// TIA Portal project "0000" (V15.1)

(* hardware
DEVICE "S7-1200-Station_1"  S7-1200 Station
   slot 0: "Baugruppenträger_0"  S7-1200 Rack  Rack  V1.0
   slot 1: "0000"  CPU 1214C DC/DC/DC  6ES7 214-1AG40-0XB0  V4.3
DEVICE "S7300/ET200M-Station_1"  S7-300 station
   slot 0: "Profilschiene_0"  Rail  6ES7 390-1***0-0AA0
   slot 2: "0001"  CPU 317-2 PN/DP  6ES7 317-2EK13-0AB0  V2.6
      slot 1: "MPI/DP-Schnittstelle_1"  X1
      slot 2: "PROFINET-Schnittstelle_1"  PN-IO
         slot 1: "Port_1"  Port
DEVICE "S71500/ET200MP-Station_1"  S7-1500 station
   slot 0: "Profilschiene_0"  Rack  6ES7 590-1***0-0AA0
   slot 1: "PLC_1"  CPU 1515-2 PN  6ES7 515-2AM01-0AB0  V2.6
      slot 3: "CPU-Display_1"  6ES7591-1BA00-0AA0
*)

// ===== PLC "0000"  CPU 1214C DC/DC/DC =====

VAR_GLOBAL   // PLC tag table "Standard-Variablentabelle"
   "Clock_Byte" AT %MB1 : Byte;
   "Clock_10Hz" AT %M1.0 : Bool;
   "Clock_5Hz" AT %M1.1 : Bool;
   "Clock_2.5Hz" AT %M1.2 : Bool;
   "Clock_2Hz" AT %M1.3 : Bool;
   "Clock_1.25Hz" AT %M1.4 : Bool;
   "Clock_1Hz" AT %M1.5 : Bool;
   "Clock_0.625Hz" AT %M1.6 : Bool;
   "Clock_0.5Hz" AT %M1.7 : Bool;
   "System_Byte" AT %MB0 : Byte;
   "FirstScan" AT %M0.0 : Bool;
   "DiagStatusUpdate" AT %M0.1 : Bool;
   "AlwaysTRUE" AT %M0.2 : Bool;
   "AlwaysFALSE" AT %M0.3 : Bool;
   "Test" AT %M10.0 : Bool;
   "Tag_1" AT %M100.0 : Bool;
   "Tag_2" AT %M100.2 : Bool;
   "Tag_3" AT %M200.0 : Bool;
   "%M200.1" AT %M200.1 : Bool;
END_VAR

TYPE "Daten"
TITLE = has no title
// some comment
   STRUCT
      Aktiv : Bool := True;   // Anlage an oder aus
      Codierung : Byte := 16#2;   // Codierung
      Status : Word := 16#FF;   // Status
      Status_erweitert : DWord := 16#FFFF;   // Erweiterter Status
      Programmnummer : Int := 3;   // Aktuelle Programmnummer
      Zaehler : DInt := 5;   // Zählerstand
      Stationsname : String := 'Anlage001';   // Name der Station
      Zeitstempel : DTL;   // Aktueller Zeitstempel
   END_STRUCT;
END_TYPE

DATA_BLOCK "ConPlc_DB"   // DB1
{ S7_Optimized_Access := 'TRUE' }
VERSION : 0.1
// stored: InstanceOfName ConPlc
"ConPlc"
BEGIN
END_DATA_BLOCK

// folder: Testdata

DATA_BLOCK "Testdata"   // DB3
{ S7_Optimized_Access := 'FALSE' }
VERSION : 0.1
   VAR
      Daten : "Daten";
   END_VAR
BEGIN
END_DATA_BLOCK

// folder: (top level)

FUNCTION_BLOCK "ConPlc"   // FB1000, SCL
{ S7_Optimized_Access := 'TRUE' }
VERSION : 0.1
   VAR_INPUT
      ACTIVATE : Bool := False;   // activate connection
      TACT : Bool := False;   // tact
      CONN_ID : Conn_Ouc := 16#1;   // connection reference / identifier
      HW_ID : Hw_Any := 64;   // HW-identifier of IE-interface submodule
      CONN_Type : Byte := 16#0B;   // type of connection: 11=TCP/IP, 19=UDP (17=TCP/IP)
      IP_ADDR_1 : Byte := 16#C0;   // IPv4 address
      IP_ADDR_2 : Byte := 16#A8;   // IPv4 address
      IP_ADDR_3 : Byte := 16#00;   // IPv4 address
      IP_ADDR_4 : Byte := 16#1E;   // IPv4 address
      PORT_Remote : UInt := 2000;   // remote UDP/TCP port number
      PORT_Local : UInt := 2000;   // local UDP/TCP port number
   END_VAR
   VAR_IN_OUT
      DATA : Variant;
   END_VAR
   VAR
      ACT_CONN : Bool;
      CONN_ESTABLISHED : Bool;
      DONE_CONN : Bool;
      BUSY_CONN : Bool;
      ERROR_CONN : Bool;
      STATUS_CONN : Word;
      DONE_SEND : Bool;
      BUSY_SEND : Bool;
      ERROR_SEND : Bool;
      STATUS_SEND : Word;
      ACT_SEND : Bool;
      NDR_RECV : Bool;
      BUSY_RECV : Bool;
      ERROR_RECV : Bool;
      STATUS_RECV : Word;
      RCVD_LEN : UDInt;
      ACT_RECV : Bool;
      DONE_DISCON : Bool;
      BUSY_DISCON : Bool;
      ERROR_DISCON : Bool;
      STATUS_DISCON : Word;
      ACT_DISCON : Bool;
      TRIGGER : Bool;
      TRIGGER_MEM : Bool;
      TCON_IDB : TCON;
      TSEND_IDB : TSEND;
      TRCV_IDB : TRCV;
      TDISCON_IDB : TDISCON;
      CONN_PARAMETER : TCON_IP_v4;
      TON_RESET : TON_TIME;
   END_VAR
   // CONN_PARAMETER.InterfaceId := 64;
   // CONN_PARAMETER.ID := 16#1;
   // CONN_PARAMETER.ConnectionType := 16#0B;
   // CONN_PARAMETER.ActiveEstablished := False;
   // CONN_PARAMETER.RemoteAddress.ADDR[1] := 16#C0;
   // CONN_PARAMETER.RemoteAddress.ADDR[2] := 16#A8;
   // CONN_PARAMETER.RemoteAddress.ADDR[3] := 16#00;
   // CONN_PARAMETER.RemoteAddress.ADDR[4] := 16#1E;
   // CONN_PARAMETER.RemotePort := 2000;
   // CONN_PARAMETER.LocalPort := 2000;
BEGIN
   REGION set connection data
       #CONN_PARAMETER.ID := #CONN_ID;
       #CONN_PARAMETER.InterfaceId := #HW_ID;
       #CONN_PARAMETER.ActiveEstablished := TRUE;
       #CONN_PARAMETER.ConnectionType := #CONN_Type;
       #CONN_PARAMETER.RemoteAddress.ADDR[1] := #IP_ADDR_1;
       #CONN_PARAMETER.RemoteAddress.ADDR[2] := #IP_ADDR_2;
       #CONN_PARAMETER.RemoteAddress.ADDR[3] := #IP_ADDR_3;
       #CONN_PARAMETER.RemoteAddress.ADDR[4] := #IP_ADDR_4;
       #CONN_PARAMETER.RemotePort := #PORT_Remote;
       #CONN_PARAMETER.LocalPort := #PORT_Local;
   END_REGION

   REGION create trigger
       #TRIGGER := #TACT AND NOT #TRIGGER_MEM;
       #TRIGGER_MEM := #TACT;
   END_REGION

   REGION connect
       //connect enable
       IF #ACTIVATE AND NOT #CONN_ESTABLISHED THEN
           #ACT_CONN := True;
       END_IF;
       //connect
       #TCON_IDB(REQ       := #ACT_CONN AND #TRIGGER,
                 ID        := #CONN_ID,
                 DONE      => #DONE_CONN,
                 BUSY      => #BUSY_CONN,
                 ERROR     => #ERROR_CONN,
                 STATUS    => #STATUS_CONN,
                 CONNECT   := #CONN_PARAMETER);
       //connect done
       IF #DONE_CONN THEN
           #CONN_ESTABLISHED := True;
           #ACT_CONN := False;
       END_IF;
   END_REGION

   REGION send
       //send enable
       #ACT_SEND := #CONN_ESTABLISHED AND #TRIGGER AND NOT #BUSY_SEND;
       //send
       #TSEND_IDB(REQ      := #ACT_SEND,
                  ID       := #CONN_ID,
                  LEN      := 0,
                  DONE     => #DONE_SEND,
                  BUSY     => #BUSY_SEND,
                  ERROR    => #ERROR_SEND,
                  STATUS   => #STATUS_SEND,
                  DATA     := #DATA);
   END_REGION

   // REGION recieve
   //     //revieve enable
   //     #ACT_RECV := #CONN_ESTABLISHED;
   //     //recieve
   //     #TRCV_IDB(EN_R      := #ACT_RECV,
   //               ID        := #CONN_ID,
   //               LEN       := 0,
   //               ADHOC     := FALSE,
   //               NDR       => #NDR_RECV,
   //               BUSY      => #BUSY_RECV,
   //               ERROR     => #ERROR_RECV,
   //               STATUS    => #STATUS_RECV,
   //               RCVD_LEN  => #RCVD_LEN,
   //               DATA      := #DATA);
   // END_REGION

   REGION disconnect
       //disconnect enable
       #TON_RESET(IN := #ACTIVATE AND NOT #CONN_ESTABLISHED,
                  PT := T#5s);
       #ACT_DISCON := (#TON_RESET.Q) OR (NOT #ACTIVATE);
       //disconnect
       #TDISCON_IDB(REQ    := #ACT_DISCON,
                    ID     := #CONN_ID,
                    DONE   => #DONE_DISCON,
                    BUSY   => #BUSY_DISCON,
                    ERROR  => #ERROR_DISCON,
                    STATUS => #STATUS_DISCON);

       //disconnect done
       IF NOT #ACTIVATE THEN
           #CONN_ESTABLISHED := False;
           #ACT_CONN := False;
       END_IF;
   END_REGION
END_FUNCTION_BLOCK

ORGANIZATION_BLOCK "Main"   // OB1, FBD, ProgramCycle
TITLE = "Main Program Sweep (Cycle)"
{ S7_Optimized_Access := 'TRUE' }
VERSION : 0.1
   VAR_INPUT
      Initial_Call : Bool;   // Initial call of this OB
      Remanence : Bool;   // =True, if remanent data are available
   END_VAR
   VAR_TEMP
      retval : Int;
   END_VAR
BEGIN

REGION Network 1
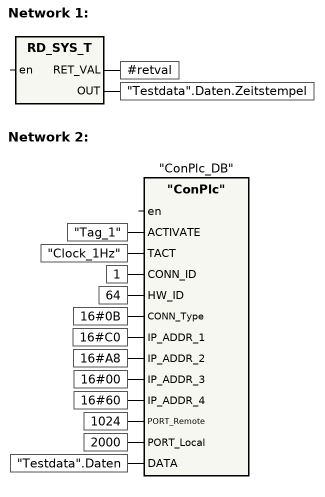
   #retval := RD_SYS_T(OUT => "Testdata".Daten.Zeitstempel);
END_REGION

REGION Network 2
   "ConPlc_DB"(ACTIVATE := "Tag_1",   // "ConPlc"
               TACT := "Clock_1Hz",
               CONN_ID := 1,
               HW_ID := 64,
               CONN_Type := 16#0B,
               IP_ADDR_1 := 16#C0,
               IP_ADDR_2 := 16#A8,
               IP_ADDR_3 := 16#00,
               IP_ADDR_4 := 16#60,
               PORT_Remote := 1024,
               PORT_Local := 2000,
               DATA := "Testdata".Daten);
END_REGION
END_ORGANIZATION_BLOCK

// ===== PLC "0001"  CPU 317-2 PN/DP =====

VAR_GLOBAL   // PLC tag table "Standard-Variablentabelle"
   "Test" AT %M10.0 : Bool;
   "Clock_Byte" AT %MB0 : Byte;
   "Clock_10Hz" AT %M0.0 : Bool;
   "Clock_5Hz" AT %M0.1 : Bool;
   "Clock_2.5Hz" AT %M0.2 : Bool;
   "Clock_2Hz" AT %M0.3 : Bool;
   "Clock_1.25Hz" AT %M0.4 : Bool;
   "Clock_1Hz" AT %M0.5 : Bool;
   "Clock_0.625Hz" AT %M0.6 : Bool;
   "Clock_0.5Hz" AT %M0.7 : Bool;
END_VAR

ORGANIZATION_BLOCK "Main"   // OB1, SCL
TITLE = "Main Program Sweep (Cycle)"
{ S7_Optimized_Access := 'FALSE' }
VERSION : 0.1
   VAR_TEMP
      OB1_EV_CLASS : Byte;   // Bits 0-3 = 1 (Coming event), Bits 4-7 = 1 (Event class 1)
      OB1_SCAN_1 : Byte;   // 1 (Cold restart scan 1 of OB 1), 3 (Scan 2-n of OB 1)
      OB1_PRIORITY : Byte;   // Priority of OB Execution
      OB1_OB_NUMBR : Byte;   // 1 (Organization block 1, OB1)
      OB1_RESERVED_1 : Byte;   // Reserved for system
      OB1_RESERVED_2 : Byte;   // Reserved for system
      OB1_PREV_CYCLE : Int;   // Cycle time of previous OB1 scan (milliseconds)
      OB1_MIN_CYCLE : Int;   // Minimum cycle time of OB1 (milliseconds)
      OB1_MAX_CYCLE : Int;   // Maximum cycle time of OB1 (milliseconds)
      OB1_DATE_TIME : Date_And_Time;   // Date and time OB1 started
   END_VAR
BEGIN
   REGION Test
       "Test" := "Clock_0.5Hz";
   END_REGION
END_ORGANIZATION_BLOCK

// ===== PLC "PLC_1"  CPU 1515-2 PN =====

FUNCTION_BLOCK "S7-1500_CPU_Comm_TCP_master"   // FB250, STL
TITLE = FB to master connection to partner CPU
{ S7_Optimized_Access := 'FALSE' }
VERSION : 0.1
   VAR_INPUT
      CONN_stop : Bool := False;   // stop connection
      Takt : Bool := False;
      CONN_ID : Conn_Ouc := 16#1;   // connection reference / identifier
      HW_ID : Hw_Any := 64;   // HW-identifier of IE-interface submodule
      CONN_Type : Byte := 16#0B;   // type of connection: 11=TCP/IP, 19=UDP (17=TCP/IP)
      IP_ADDR_1 : Byte := 16#C0;   // IPv4 address
      IP_ADDR_2 : Byte := 16#A8;   // IPv4 address
      IP_ADDR_3 : Byte := 16#00;   // IPv4 address
      IP_ADDR_4 : Byte := 16#1E;   // IPv4 address
      remote_port : UInt := 2000;   // remote UDP/TCP port number
      local_port : UInt := 2000;   // local UDP/TCP port number
   END_VAR
   VAR
      START_CONN : Bool;
      CONN_established : Bool;
      DONE_CONN : Bool;
      BUSY_CONN : Bool;
      ERROR_CONN : Bool;
      STATUS_CONN : Word;
      DONE_SEND : Bool;
      BUSY_SEND : Bool;
      ERROR_SEND : Bool;
      STATUS_SEND : Word;
      ACT_SEND : Bool;
      NDR_RECV : Bool;
      BUSY_RECV : Bool;
      ERROR_RECV : Bool;
      STATUS_RECV : Word;
      RCVD_LEN : UDInt;
      DONE_DISCON : Bool;
      BUSY_DISCON : Bool;
      ERROR_DISCON : Bool;
      STATUS_DISCON : Word;
      TCON_IDB : TCON;
      TSEND_IDB : TSEND;
      TRCV_IDB : TRCV;
      TDISCON_IDB : TDISCON;
      CONN_parameter : TCON_IP_v4;
      SEND_DATA : Struct
         Lebensbit : Bool;
         Störung_Vakuum : Bool;
         Reserve_bit_2 : Bool;
         Reserve_bit_3 : Bool;
         Reserve_bit_4 : Bool;
         Reserve_bit_5 : Bool;
         Reserve_bit_6 : Bool;
         Reserve_bit_7 : Bool;
         Temperatur : Int := 20;   // Umgebungstemperatur in °C
         Absolutdruck : Int := 1000;   // Absolutdruck in mbar
      END_STRUCT;
      RECV_DATA : Struct
         Lebensbit : Bool;
         Reserve_bit_1 : Bool;
         Reserve_bit_2 : Bool;
         Reserve_bit_3 : Bool;
         Reserve_bit_4 : Bool;
         Reserve_bit_5 : Bool;
         Reserve_bit_6 : Bool;
         Reserve_bit_7 : Bool;
      END_STRUCT;
   END_VAR
   VAR_TEMP
      conn_trigger : Bool;
   END_VAR
   // CONN_parameter.InterfaceId := 64;
   // CONN_parameter.ID := 16#1;
   // CONN_parameter.ConnectionType := 16#0B;
   // CONN_parameter.ActiveEstablished := False;
   // CONN_parameter.RemotePort := 2000;
   // CONN_parameter.LocalPort := 2000;
   // CONN_parameter.RemoteAddress.ADDR[1] := 16#C0;
   // CONN_parameter.RemoteAddress.ADDR[2] := 16#A8;
   // CONN_parameter.RemoteAddress.ADDR[3] := 16#00;
   // CONN_parameter.RemoteAddress.ADDR[4] := 16#1E;
BEGIN

REGION Network 1: set connection data
   //---------------------------------
         L     #CONN_ID;
         T     #CONN_parameter.ID;
   //---------------------------------
         L     #HW_ID;
         T     #CONN_parameter.InterfaceId;
   //---------------------------------
         SET;  //Master wartet das sich der slave meldet
         R     #CONN_parameter.ActiveEstablished;
   //---------------------------------
         L     #CONN_Type;
         T     #CONN_parameter.ConnectionType;
   //---------------------------------
         L     #IP_ADDR_1;
         T     #CONN_parameter.RemoteAddress.ADDR[1];
         L     #IP_ADDR_2;
         T     #CONN_parameter.RemoteAddress.ADDR[2];
         L     #IP_ADDR_3;
         T     #CONN_parameter.RemoteAddress.ADDR[3];
         L     #IP_ADDR_4;
         T     #CONN_parameter.RemoteAddress.ADDR[4];
   //---------------------------------
         L     #remote_port;
         T     #CONN_parameter.RemotePort;
   //---------------------------------
         L     #local_port;
         T     #CONN_parameter.LocalPort;
   //---------------------------------
END_REGION

REGION Network 2: start connect
         A(;
         AN    #CONN_established;
         AN    #CONN_stop;
         );
         S     #START_CONN;
END_REGION

REGION Network 3: connect
         A     #START_CONN;
         =     #conn_trigger;

         CALL  #TCON_IDB
         ( REQ     := #conn_trigger,
           ID      := #CONN_ID,
           DONE    := #DONE_CONN,
           BUSY    := #BUSY_CONN,
           ERROR   := #ERROR_CONN,
           STATUS  := #STATUS_CONN,
           CONNECT := #CONN_parameter
         );
END_REGION

REGION Network 4: done connect
         A     #DONE_CONN;
         S     #CONN_established;
         R     #START_CONN;
END_REGION

REGION Network 5: automaticly trigger send data if sending is not active anymore
         AN    #BUSY_SEND;
         A     #Takt;
         =     #ACT_SEND;
END_REGION

REGION Network 6: send
         CALL  #TSEND_IDB
         ( REQ    := #ACT_SEND,
           ID     := #CONN_ID,
           LEN    := 0,
           DONE   := #DONE_SEND,
           BUSY   := #BUSY_SEND,
           ERROR  := #ERROR_SEND,
           STATUS := #STATUS_SEND,
           DATA   := #SEND_DATA
         );
END_REGION

REGION Network 7: recieve
         CALL  #TRCV_IDB
         ( EN_R     := #CONN_established,
           ID       := #CONN_ID,
           LEN      := 0,
           ADHOC    := FALSE,
           NDR      := #NDR_RECV,
           BUSY     := #BUSY_RECV,
           ERROR    := #ERROR_RECV,
           STATUS   := #STATUS_RECV,
           RCVD_LEN := #RCVD_LEN,
           DATA     := #RECV_DATA
         );
END_REGION

REGION Network 8: disconnect
         A     #CONN_stop;
         R     #CONN_established;
         R     #START_CONN;

         CALL  #TDISCON_IDB
         ( REQ    := #CONN_stop,
           ID     := #CONN_ID,
           DONE   := #DONE_DISCON,
           BUSY   := #BUSY_DISCON,
           ERROR  := #ERROR_DISCON,
           STATUS := #STATUS_DISCON
         );
END_REGION
END_FUNCTION_BLOCK

FUNCTION_BLOCK "S7-1500_CPU_Comm_TCP_slave"   // FB251, STL
TITLE = FB to slave connection to partner CPU
{ S7_Optimized_Access := 'FALSE' }
VERSION : 0.1
   VAR_INPUT
      CONN_stop : Bool := False;   // stop connection
      Takt : Bool := False;
      CONN_ID : Conn_Ouc := 16#1;   // connection reference / identifier
      HW_ID : Hw_Any := 64;   // HW-identifier of IE-interface submodule
      CONN_Type : Byte := 16#0B;   // type of connection: 11=TCP/IP, 19=UDP (17=TCP/IP)
      IP_ADDR_1 : Byte := 16#C0;   // IPv4 address
      IP_ADDR_2 : Byte := 16#A8;   // IPv4 address
      IP_ADDR_3 : Byte := 16#00;   // IPv4 address
      IP_ADDR_4 : Byte := 16#1E;   // IPv4 address
      remote_port : UInt := 2000;   // remote UDP/TCP port number
      local_port : UInt := 2000;   // local UDP/TCP port number
   END_VAR
   VAR
      START_CONN : Bool;
      CONN_established : Bool;
      DONE_CONN : Bool;
      BUSY_CONN : Bool;
      ERROR_CONN : Bool;
      STATUS_CONN : Word;
      DONE_SEND : Bool;
      BUSY_SEND : Bool;
      ERROR_SEND : Bool;
      STATUS_SEND : Word;
      ACT_SEND : Bool;
      NDR_RECV : Bool;
      BUSY_RECV : Bool;
      ERROR_RECV : Bool;
      STATUS_RECV : Word;
      RCVD_LEN : UDInt;
      DONE_DISCON : Bool;
      BUSY_DISCON : Bool;
      ERROR_DISCON : Bool;
      STATUS_DISCON : Word;
      TCON_IDB : TCON;
      TSEND_IDB : TSEND;
      TRCV_IDB : TRCV;
      TDISCON_IDB : TDISCON;
      CONN_parameter : TCON_IP_v4;
      SEND_DATA : Struct
         Lebensbit : Bool;
         Reserve_bit_1 : Bool;
         Reserve_bit_2 : Bool;
         Reserve_bit_3 : Bool;
         Reserve_bit_4 : Bool;
         Reserve_bit_5 : Bool;
         Reserve_bit_6 : Bool;
         Reserve_bit_7 : Bool;
      END_STRUCT;
      RECV_DATA : Struct
         Lebensbit : Bool;
         Störung_Vakuum : Bool;
         Reserve_bit_2 : Bool;
         Reserve_bit_3 : Bool;
         Reserve_bit_4 : Bool;
         Reserve_bit_5 : Bool;
         Reserve_bit_6 : Bool;
         Reserve_bit_7 : Bool;
         Temperatur : Int := 20;   // Umgebungstemperatur in °C
         Absolutdruck : Int := 1000;   // Absolutdruck in mbar
      END_STRUCT;
   END_VAR
   VAR_TEMP
      conn_trigger : Bool;
   END_VAR
   // CONN_parameter.InterfaceId := 64;
   // CONN_parameter.ID := 16#1;
   // CONN_parameter.ConnectionType := 16#0B;
   // CONN_parameter.ActiveEstablished := False;
   // CONN_parameter.RemotePort := 2000;
   // CONN_parameter.LocalPort := 2000;
   // CONN_parameter.RemoteAddress.ADDR[1] := 16#C0;
   // CONN_parameter.RemoteAddress.ADDR[2] := 16#A8;
   // CONN_parameter.RemoteAddress.ADDR[3] := 16#00;
   // CONN_parameter.RemoteAddress.ADDR[4] := 16#1E;
BEGIN

REGION Network 1: xxxset connection data
   //---------------------------------
         L     #CONN_ID;
         T     #CONN_parameter.ID;
   //---------------------------------
         L     #HW_ID;
         T     #CONN_parameter.InterfaceId;
   //---------------------------------
         SET;  //Slave versucht aktiv die verbindung aufzubauen
         S     #CONN_parameter.ActiveEstablished;
   //---------------------------------
         L     #CONN_Type;
         T     #CONN_parameter.ConnectionType;
   //---------------------------------
         L     #IP_ADDR_1;
         T     #CONN_parameter.RemoteAddress.ADDR[1];
         L     #IP_ADDR_2;
         T     #CONN_parameter.RemoteAddress.ADDR[2];
         L     #IP_ADDR_3;
         T     #CONN_parameter.RemoteAddress.ADDR[3];
         L     #IP_ADDR_4;
         T     #CONN_parameter.RemoteAddress.ADDR[4];
   //---------------------------------
         L     #remote_port;
         T     #CONN_parameter.RemotePort;
   //---------------------------------
         L     #local_port;
         T     #CONN_parameter.LocalPort;
   //---------------------------------
END_REGION

REGION Network 2: xxxstart connect
         A(;
         AN    #CONN_established;
         AN    #CONN_stop;
         );
         S     #START_CONN;
END_REGION

REGION Network 3: xxxconnect
         A     #START_CONN;
         A     #Takt;
         =     #conn_trigger;

         CALL  #TCON_IDB
         ( REQ     := #conn_trigger,
           ID      := #CONN_ID,
           DONE    := #DONE_CONN,
           BUSY    := #BUSY_CONN,
           ERROR   := #ERROR_CONN,
           STATUS  := #STATUS_CONN,
           CONNECT := #CONN_parameter
         );
END_REGION

REGION Network 4: xxxdone connect
         A     #DONE_CONN;
         S     #CONN_established;
         R     #START_CONN;
END_REGION

REGION Network 5: automaticly trigger send data if new data recieved
         A     #NDR_RECV;
         =     #ACT_SEND;
END_REGION

REGION Network 6: send
         CALL  #TSEND_IDB
         ( REQ    := #ACT_SEND,
           ID     := #CONN_ID,
           LEN    := 0,
           DONE   := #DONE_SEND,
           BUSY   := #BUSY_SEND,
           ERROR  := #ERROR_SEND,
           STATUS := #STATUS_SEND,
           DATA   := #SEND_DATA
         );
END_REGION

REGION Network 7: recieve
         CALL  #TRCV_IDB
         ( EN_R     := #CONN_established,
           ID       := #CONN_ID,
           LEN      := 0,
           ADHOC    := FALSE,
           NDR      := #NDR_RECV,
           BUSY     := #BUSY_RECV,
           ERROR    := #ERROR_RECV,
           STATUS   := #STATUS_RECV,
           RCVD_LEN := #RCVD_LEN,
           DATA     := #RECV_DATA
         );
END_REGION

REGION Network 8: disconnect
         A     #CONN_stop;
         R     #CONN_established;
         R     #START_CONN;

         CALL  #TDISCON_IDB
         ( REQ    := #CONN_stop,
           ID     := #CONN_ID,
           DONE   := #DONE_DISCON,
           BUSY   := #BUSY_DISCON,
           ERROR  := #ERROR_DISCON,
           STATUS := #STATUS_DISCON
         );
END_REGION
END_FUNCTION_BLOCK

FUNCTION "SPS-Kommunikation" : Void   // FC250, STL
TITLE = Kommunikation mit anderer CPU aufbauen
{ S7_Optimized_Access := 'TRUE' }
VERSION : 0.1
   VAR_TEMP
      connection_stop : Bool;
   END_VAR
BEGIN

REGION Network 1: Daten rangieren
         L     "DB350_Umgebungseinflüsse".Temperatur;
         T     "S7-1500_CPU_Comm_TCP_master_DB".SEND_DATA.Temperatur;

         L     "DB350_Umgebungseinflüsse".Absolutdruck;
         T     "S7-1500_CPU_Comm_TCP_master_DB".SEND_DATA.Absolutdruck;

         A     "Störung_Vakuum";
         =     "S7-1500_CPU_Comm_TCP_master_DB".SEND_DATA.Störung_Vakuum;
END_REGION

REGION Network 2: Lebensbit mit Takt an Partner senden, Lebensbit von Partner überwachen
         A     "Clock_1Hz";
         =     "S7-1500_CPU_Comm_TCP_master_DB".SEND_DATA.Lebensbit;

         A     "ME_STSP_EIN";
         A     "S7-1500_CPU_Comm_TCP_master_DB".RECV_DATA.Lebensbit;
         L     s5t#10s;
         SD    "T-CPU-CPU_Comm_Error_01";

         A     "ME_STSP_EIN";
         AN    "S7-1500_CPU_Comm_TCP_master_DB".RECV_DATA.Lebensbit;
         L     s5t#10s;
         SD    "T-CPU-CPU_Comm_Error_02";
END_REGION

REGION Network 3: Kommunikationsaufruf
         A     "ME_STSP_EIN";
         L     s5t#3s;
         SE    "T-comm_restart";

         A     "T-comm_restart";
         =     #connection_stop;

   //CPU mit aktiven Verbindungsaufbau
         CALL  "S7-1500_CPU_Comm_TCP_master", "S7-1500_CPU_Comm_TCP_master_DB"
         ( CONN_stop   := #connection_stop,  //Stoppen der Verbindung
           Takt        := "Clock_0.5Hz",  //Taktsignal
           CONN_ID     := 5,
           HW_ID       := 64,  //HW-ID der Profinet Schnittstelle (in diesem Beispiel [X1])
           CONN_Type   := 16#0B,  //Steht für TCP verbindungsart
           IP_ADDR_1   := 16#C0,  //192 IP-Adresse der Partner CPU
           IP_ADDR_2   := 16#A8,  //168
           IP_ADDR_3   := 16#00,  //0
           IP_ADDR_4   := 16#04,  //4
           remote_port := 2000,  //partner Portnummer
           local_port  := 2000  //eigene Portnummer
         );
END_REGION
END_FUNCTION

FUNCTION "SPS-Kommunikation_1" : Void   // FC250, STL
TITLE = Kommunikation mit anderer CPU aufbauen
{ S7_Optimized_Access := 'TRUE' }
VERSION : 0.1
   VAR_TEMP
      connection_stop : Bool;
   END_VAR
BEGIN

REGION Network 1: Daten rangieren
         L     "S7-1500_CPU_Comm_TCP_slave_DB".RECV_DATA.Temperatur;
         T     "DB350_Umgebungseinflüsse".Temperatur;

         L     "S7-1500_CPU_Comm_TCP_slave_DB".RECV_DATA.Absolutdruck;
         T     "DB350_Umgebungseinflüsse".Absolutdruck;

         A     "S7-1500_CPU_Comm_TCP_slave_DB".RECV_DATA.Störung_Vakuum;
         =     "Störung_Vakuum";
END_REGION

REGION Network 2: Lebensbit mit Takt an Partner senden, Lebensbit von Partner überwachen
         A     "Clock_1Hz";
         =     "S7-1500_CPU_Comm_TCP_slave_DB".SEND_DATA.Lebensbit;

         A     "ME_STSP_EIN";
         A     "S7-1500_CPU_Comm_TCP_slave_DB".RECV_DATA.Lebensbit;
         L     s5t#10s;
         SD    "T-CPU-CPU_Comm_Error_01";

         A     "ME_STSP_EIN";
         AN    "S7-1500_CPU_Comm_TCP_slave_DB".RECV_DATA.Lebensbit;
         L     s5t#10s;
         SD    "T-CPU-CPU_Comm_Error_02";
END_REGION

REGION Network 3: Kommunikationsaufruf
         A     "ME_STSP_EIN";
         L     s5t#3s;
         SE    "T-comm_restart";

         A     "T-comm_restart";
         =     #connection_stop;

   //CPU mit Passivem Verbindungsaufbau
         CALL  "S7-1500_CPU_Comm_TCP_slave", "S7-1500_CPU_Comm_TCP_slave_DB"
         ( CONN_stop   := #connection_stop,  //Stoppen der Verbindung
           Takt        := "Clock_0.5Hz",  //Taktsignal
           CONN_ID     := 5,  //verbindungsnummer (darf nur einmal vergeben werden)
           HW_ID       := 64,  //HW-ID der Profinet Schnittstelle (in diesem Beispiel [X2])
           CONN_Type   := 16#0B,  //Steht für TCP verbindungsart
           IP_ADDR_1   := 16#C0,  //192 IP-Adresse der Partner CPU
           IP_ADDR_2   := 16#A8,  //168
           IP_ADDR_3   := 16#00,  //0
           IP_ADDR_4   := 16#02,  //2
           remote_port := 2000,  //partner Portnummer
           local_port  := 2000  //eigene Portnummer
         );
END_REGION
END_FUNCTION

ORGANIZATION_BLOCK "Main"   // OB1, LAD, ProgramCycle
TITLE = "Main Program Sweep (Cycle)"
{ S7_Optimized_Access := 'TRUE' }
VERSION : 0.1
   VAR_INPUT
      Initial_Call : Bool;   // Initial call of this OB
      Remanence : Bool;   // =True, if remanent data are available
   END_VAR
BEGIN
END_ORGANIZATION_BLOCK